// Mitsubishi GX Works2 project: IELET2103_Datalab2_Oppg2   PLC: FX2N/FX2NC
// IELET2103_Datalab2_Oppg2

// task Task_01 (event TRUE, interval 0, priority 31): Oppgave2c)

PROGRAM Oppgave2a)
(* structured ladder/FBD written out as ST: instructions are called as NAME(EN, inputs, outputs); _pN, _eN, _tN stand for wires *)
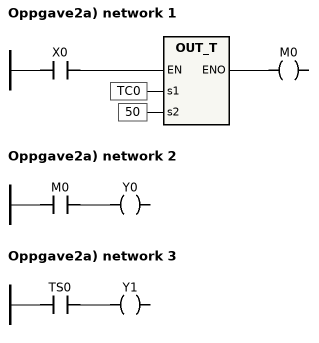
(* network 1 *)
_e1 := OUT_T(X0, TC0, 50);
M0 := _e1;
(* network 2 *)
Y0 := M0;
(* network 3 *)
Y1 := TS0;
END_PROGRAM

PROGRAM Oppgave2b)
(* structured ladder/FBD written out as ST: instructions are called as NAME(EN, inputs, outputs); _pN, _eN, _tN stand for wires *)
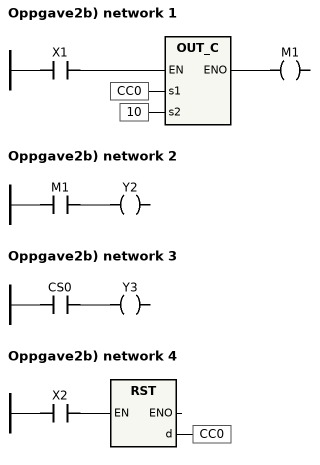
(* network 1 *)
_e1 := OUT_C(X1, CC0, 10);
M1 := _e1;
(* network 2 *)
Y2 := M1;
(* network 3 *)
Y3 := CS0;
(* network 4 *)
RST(X2, CC0);
END_PROGRAM

PROGRAM Oppgave2c)
(* structured ladder/FBD written out as ST: instructions are called as NAME(EN, inputs, outputs); _pN, _eN, _tN stand for wires *)
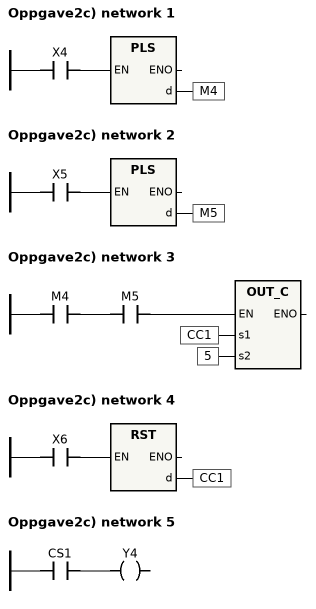
(* network 1 *)
PLS(X4, M4);
(* network 2 *)
PLS(X5, M5);
(* network 3 *)
OUT_C(M4 AND M5, CC1, 5);
(* network 4 *)
RST(X6, CC1);
(* network 5 *)
Y4 := CS1;
END_PROGRAM
